Yaskawa INFORM job: R1_W60,62(0,0)KM-OK.JBI

/JOB
//NAME R1_W60,62(0,0)KM-OK
///FOLDERNAME KRIS-SCIANA
//POS
///NPOS 52,52,0,3,0,0
///TOOL 0
///POSTYPE PULSE
///PULSE
C00000=13636,99636,9780,-8654,98943,76429
C00001=-108489,-114731,-83969,20163,84240,7679
C00002=-192773,-114731,-83969,20163,84240,7679
C00003=-195814,-97363,-54861,18109,45254,4013
C00004=-195342,-89844,-49219,17779,45528,4291
C00005=-194075,-84778,-45529,17107,45584,4897
C00006=-193609,-83033,-44294,16854,45621,5123
C00007=-195171,-86889,-46918,17671,45590,4384
C00008=-200847,-72759,-43797,19945,61650,2720
C00009=-201427,-70884,-41989,20114,61648,2491
C00010=-199143,-72536,-44097,19526,61527,3376
C00011=-199513,-75125,-46608,19573,61817,3281
C00012=-200501,-81674,-52788,19719,62464,3007
C00013=-78280,-117024,-65873,-65050,51337,51954
C00014=231366,-50529,-85532,-14348,118547,17853
C00015=231331,-51716,-35505,-12276,87907,21200
C00016=229315,-48570,-29966,-12403,85849,20709
C00017=228522,-47247,-27691,-12456,85024,20518
C00018=228691,-45242,-25520,-12451,84753,20603
C00019=228522,-47247,-27691,-12456,85024,20518
C00020=198450,-86467,-40298,21305,45876,18510
C00021=197664,-84651,-38990,21547,46188,18217
C00022=199928,-86071,-39510,20852,45254,19054
C00023=200123,-88829,-42015,20735,45324,19162
C00024=200648,-95812,-48167,20467,45386,19423
C00025=231366,-50529,-85532,-14348,118547,17853
C00026=-78280,-117024,-65873,-65050,51337,51954
C00027=-213311,-49604,17633,63554,23884,-37086
C00028=-213325,-63096,-3307,52877,27157,-31811
C00029=-184039,-61900,-6514,-29982,24943,3423
C00030=-184658,-49771,4115,-29774,24480,3211
C00031=-208526,-45976,20499,62282,21477,-35409
C00032=-208288,-49261,17048,61233,21571,-34854
C00033=-165081,-44351,28586,-60622,23883,22376
C00034=-157100,-40029,38338,-68116,25967,28113
C00035=-149547,-33615,49878,-73667,28155,33010
C00036=-147633,-33207,51281,-74248,28827,33869
C00037=-145370,-31178,54549,-75183,29556,35026
C00038=-148980,-60645,16059,-62194,31209,27271
C00039=-144413,-93486,-26442,-51146,38697,22396
C00040=-78280,-117024,-65873,-65050,51337,51954
C00041=204216,-84591,-49290,-51682,73827,23894
C00042=222529,-60204,-40854,-53258,59442,13043
C00043=209838,-69593,-64372,-21387,53614,7801
C00044=205629,-64517,-54244,-19958,49151,6845
C00045=224696,-55460,-38333,-53253,61230,13186
C00046=224153,-56614,-39635,-53066,61047,12972
C00047=201120,-72746,-51210,-19026,42314,6129
C00048=201421,-67850,-43493,-25563,56499,3643
C00049=209436,-70972,-61365,-25883,67483,4322
C00050=228633,-84332,-87971,-29537,82290,8189
C00051=199935,-84332,-95461,-29537,82290,8189
BC00000=155408,72464,1039262
BC00001=369733,7282,784079
BC00002=369733,7282,558994
BC00003=396813,15,501820
BC00004=396813,15,501820
BC00005=396813,15,501820
BC00006=396813,15,501820
BC00007=396813,15,501820
BC00008=396812,16,501817
BC00009=396813,15,501820
BC00010=396813,15,501820
BC00011=396813,15,501820
BC00012=396813,15,501820
BC00013=398174,15,1075175
BC00014=398174,29742,582568
BC00015=398174,29742,582568
BC00016=398174,29742,582568
BC00017=398174,29742,582568
BC00018=398174,29742,582568
BC00019=398174,29742,582568
BC00020=398174,29742,582568
BC00021=398174,29742,582568
BC00022=398174,29742,582568
BC00023=398174,29742,582568
BC00024=398174,29742,582568
BC00025=398174,29742,582568
BC00026=398174,15,1075175
BC00027=389408,15,893628
BC00028=389408,15,786093
BC00029=382985,15,771596
BC00030=382985,15,771596
BC00031=382985,15,771598
BC00032=382985,15,771598
BC00033=382985,15,771596
BC00034=382986,15,771595
BC00035=382986,15,771595
BC00036=382986,15,771595
BC00037=382986,15,771595
BC00038=382986,15,771595
BC00039=382986,15,771595
BC00040=398174,15,1075175
BC00041=344180,85519,956119
BC00042=398174,101082,597796
BC00043=398174,92745,477780
BC00044=398174,92745,477780
BC00045=398174,92745,477780
BC00046=398174,92745,477780
BC00047=398174,92745,477780
BC00048=398174,92745,477780
BC00049=398174,92745,477780
BC00050=398174,92745,477780
BC00051=398174,92745,562444
///POSTYPE BASE
///RECTAN
///RCONF 0,0,0,0,1,0,0,0,0,0,0,0,0,0,0,0,0,0,0,0,0,0,0,0
P00006=2.006,1.622,-0.565,0.0000,0.0000,0.0000
P00021=0.073,2.058,-0.109,0.0000,0.0000,0.0000
///RCONF 0,0,0,0,0,0,0,0,0,0,0,0,0,0,0,0,0,0,0,0,0,0,0,0
P00023=-2.957,-4.083,2.762,0.0000,0.0000,0.0000
//INST
///DATE 2023/12/07 18:16
///ATTR SC,RW
///GROUP1 RB1,BS1
NOP
'r1_W60,62(0,0)
'Path S1540 (for W415)
SFTOF
MOVJ C00000 BC00000 VJ=60.00
MOVJ C00001 BC00001 VJ=60.00
MOVJ C00002 BC00002 VJ=60.00
MOVJ C00003 BC00003 VJ=60.00
MOVJ C00004 BC00004 VJ=60.00
MOVL C00005 BC00005 V=60.0
REFP 3 C00006 BC00006
CALL JOB:SEARCH-R1
SET P021 P006
SFTON P021
MOVL C00007 BC00007 V=60.0
MOVL C00008 BC00008 V=60.0
REFP 3 C00009 BC00009
CALL JOB:SEARCH-R1
SET P021 P006
SFTON P021
MOVL C00010 BC00010 V=60.0
MOVL C00011 BC00011 V=166.7
MOVL C00012 BC00012 V=166.7
'obrot 180
'Path VIA1544
SFTOF
MOVJ C00013 BC00013 VJ=60.00
'Path VIA1545
SFTOF
MOVJ C00014 BC00014 VJ=60.00
'Path S1546 (for W18)
SFTOF
MOVJ C00015 BC00015 VJ=60.00
MOVJ C00016 BC00016 VJ=60.00
MOVL C00017 BC00017 V=60.0
REFP 3 C00018 BC00018
CALL JOB:SEARCH-R1
SET P023 P006
SFTON P023
MOVL C00019 BC00019 V=60.0
MOVL C00020 BC00020 V=60.0
REFP 3 C00021 BC00021
CALL JOB:SEARCH-R1
SET P023 P006
SFTON P023
MOVL C00022 BC00022 V=60.0
MOVL C00023 BC00023 V=166.7
MOVL C00024 BC00024 V=166.7
'Path VIA1548
SFTOF
MOVJ C00025 BC00025 VJ=60.00
'Path VIA1549
SFTOF
MOVJ C00026 BC00026 VJ=60.00
'Path W1550
SFTOF
SFTON P021
MOVJ C00027 BC00027 VJ=60.00
MOVJ C00028 BC00028 VJ=60.00
MOVJ C00029 BC00029 VJ=60.00
MOVL C00030 BC00030 V=100.0 PL=0
REFP 1 C00031 BC00031
REFP 2 C00032 BC00032
MACRO1 MJ#(0) ARGF10
ARCON
MOVL C00033 BC00033 V=13.3
ARCOF
MOVL C00034 BC00034 V=25.0
ARCON
MOVL C00035 BC00035 V=13.3
MOVL C00036 BC00036 V=14.2
MOVL C00037 BC00037 V=14.2
ARCOF
MOVL C00038 BC00038 V=166.7
MOVL C00039 BC00039 V=333.3
SFTOF
SFTOF
'Path VIA1552
SFTOF
MOVJ C00040 BC00040 VJ=60.00
'Path VIA1553
SFTOF
MOVJ C00041 BC00041 VJ=60.00
'Path W1555
SFTOF
SFTON P023
MOVJ C00042 BC00042 VJ=60.00
MOVJ C00043 BC00043 VJ=60.00
MOVL C00044 BC00044 V=100.0 PL=0
REFP 1 C00045 BC00045
REFP 2 C00046 BC00046
MACRO1 MJ#(0) ARGF10
ARCON
MOVL C00047 BC00047 V=14.2
MOVL C00048 BC00048 V=14.2
ARCOF
MOVL C00049 BC00049 V=166.7
MOVL C00050 BC00050 V=166.7
MOVJ C00051 BC00051 VJ=60.00
SFTOF
END
